// TIA Portal V19 export
ORGANIZATION_BLOCK "Main"   // OB3031, LAD, ProgramCycle
TITLE = "Main Program Sweep (Cycle)"
AUTHOR : Siemens_FA_SUP
// stored: AutoNumber false, IsIECCheckEnabled true, Namespace Unit.Em2, SetENOAutomatically true
   VAR_INPUT
      Initial_Call : Bool;   // Initial call of this OB
      Remanence : Bool;   // =True, if remanent data are available
   END_VAR
   VAR_TEMP
      tempIndex : Int;   // Index of EM in the array
   END_VAR
   VAR CONSTANT
      "SimulationData.SimulationActive" : Bool := true;
   END_VAR
BEGIN

REGION Network 1: Call Equipment
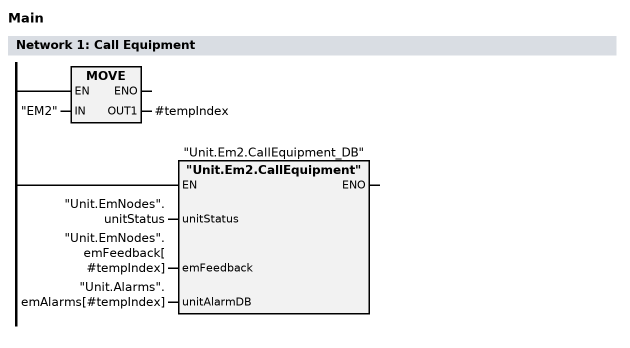
   RUNG wire#powerrail
      Move(in := "EM2", out1 => #tempIndex)
   END_RUNG
   RUNG wire#powerrail
      "Unit.Em2.CallEquipment_DB"(unitStatus := "Unit.EmNodes".unitStatus, emFeedback := "Unit.EmNodes".emFeedback[#tempIndex], unitAlarmDB := "Unit.Alarms".emAlarms[#tempIndex])
   END_RUNG
   // the same network as SCL:
   #tempIndex := "EM2";
   "Unit.Em2.CallEquipment_DB"(unitStatus := "Unit.EmNodes".unitStatus,   // "Unit.Em2.CallEquipment"
                           emFeedback := "Unit.EmNodes".emFeedback[#tempIndex],
                           unitAlarmDB := "Unit.Alarms".emAlarms[#tempIndex]);
END_REGION
END_ORGANIZATION_BLOCK
